Universal Robots PolyScope program: Example_palletsim_to_ur.urp

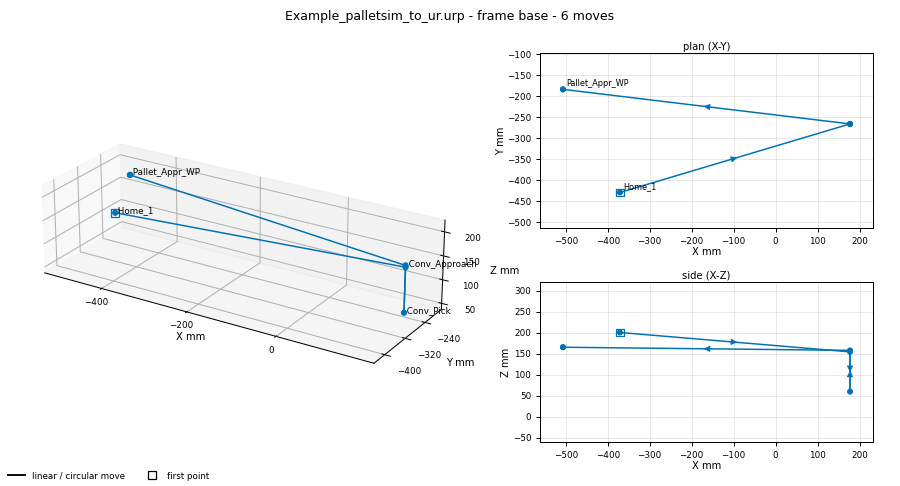
[picture p0: tool path of Example_palletsim_to_ur.urp in frame base, 6 of 9 moves have a stored position in this frame; points joined in program order, loops and branches not executed]
Program RidzwanPalletSoftware_3.2_Angle_URTrainingRoom (installation=default directory=/home/ur/ursim-current/programs createdIn=5.21.2 lastSavedIn=5.21.3 robotSerialNumber=20245799999)
Calibrated DH parameters: a=[0, -0.425, -0.3922, 0, 0, 0]; d=[0.1625, 0, 0, 0.1333, 0.0997, 0.0996]; alpha=[1.570796, 0, 0, 1.570796, -1.570796, 0]; deltaTheta=[0, 0, 0, 0, 0, 0]
InitVariablesNode
Robot Program (runOnlyOnce=false)
  Call Program_Execution
SubProgram -> Program_Execution
SubProgram Program_Execution (keepSynchronizedWithDisk=false)
  Folder Initial Instructions
    Popup Message (haltProgram=false message=Refer to the program Pop-up steps to complete the program, the following will be need/completed: <br><br> 1. IP_Address <br> 2. A.Palletizing and B. Conveyor <br> Approach and Exit waypoints <br> 3. Plane Feature  inputType=Text)
    Popup Warning (haltProgram=false message=*IMPORTANT* <br> <br> You will need to complete the instructions in all of the 'User Configuration' Folders found in the program inputType=Text)
    Popup Message (haltProgram=false message=First step will be to create a Plane Feature via the Installation tab. <br> <br> Make sure that the Origin is directly on the edge of the pallet. (Similar to visualization on Pallet Software program) inputType=Text)
  Folder Socket Configuration
    Folder User Configuration
      Popup Message (haltProgram=false message=Replace the X value below with the Manual IP_Address of the PC inputType=Text)
      PC_IPAddress := "192.168.56.5"
    Socket_Check := socket_open(PC_IPAddress,50000,socket_name="socket_0")
    asciiData := socket_read_ascii_float(8,"socket_0",timeout=0)
  MoveJ speed 60 deg/s, acceleration 80 deg/s^2 (useActiveTCP=true optimoveEnabled=false optiMoveSpeed=0.3 optiMoveAcceleration=0.09) feature=Base
    Waypoint Home_1: TCP in base x=-370.977 y=-429.532 z=201.159 mm, rx=-2.2649 ry=-2.1727 rz=-0.0079 rad; joints [-117.295, -100.067, -95.13, -75.173, 89.825, 65.225] deg; TCP offset x=0 y=0 z=176.9 mm, rx=0 ry=0 rz=0 rad
  'Conveyor'
  Folder Folder
    Folder Conveyor/Stationary Logic
      Set DigitalOutput pin=digital_out[2]; digitalValue=1
      Set AnalogOutput pin=analog_out[1]; analogValue=10
      Wait DigitalInput pin=digital_in[3]; digitalValue=1
      Wait Sleep waitTime=1
      Set DigitalOutput pin=digital_out[2]; digitalValue=0
      MoveL speed 250 mm/s, acceleration 1200 mm/s^2 (useActiveTCP=true optimoveEnabled=false optiMoveSpeed=0.3 optiMoveAcceleration=0.09) feature=Base
        Folder User Configuration
          Waypoint Conv_Approach: TCP in base x=177.389 y=-266.068 z=154.971 mm, rx=2.2689 ry=2.1729 rz=0 rad; joints [-31.936, -64.279, -132.627, -73.136, 89.936, 150.74] deg
          Waypoint Conv_Pick: TCP in base x=177.389 y=-266.068 z=60.124 mm, rx=2.2689 ry=2.1729 rz=0 rad; joints [-31.908, -72.825, -143.428, -53.79, 89.881, 150.729] deg
          Folder Gripper Logic
            URCap VG Grip (OnRobot, OnRobot A/S) dataModel(payload-weight=0.01, vg.grip.seek=false, Variable(key=on_return, variable(name=on_return)))
            Wait Sleep waitTime=0.25
          Waypoint Conv_Exit: TCP in base x=177.389 y=-266.068 z=158.52 mm, rx=2.2689 ry=2.1729 rz=0 rad; joints [-31.937, -64.094, -132.18, -73.767, 89.937, 150.74] deg
  'Pallet_Software'
  Folder Palletizing Software Logic
    boxCenterX := asciiData[3]
    boxCenterY := asciiData[4]
    AngleValue := asciiData[5]
    HeightValue := asciiData[6]
    MoveL speed 250 mm/s, acceleration 1200 mm/s^2 (useActiveTCP=true optimoveEnabled=false optiMoveSpeed=0.3 optiMoveAcceleration=0.09) feature=Base
      Folder User Configuration
        Waypoint Pallet_Appr_WP: TCP in base x=-506.661 y=-183.741 z=166.025 mm, rx=2.2689 ry=2.1729 rz=0 rad; joints [-145.856, -97.57, -103.549, -68.922, 89.882, 36.757] deg
      Wait Sleep waitTime=0.05
      tempVar := get_actual_tcp_pose()
      Pallet_App_Z := tempVar[2]
      Pallet_App_Rx := tempVar[3]
      Pallet_App_Ry := tempVar[4]
      Pallet_App_Rz := tempVar[5]
      CompilePoseRef := p[boxCenterX,boxCenterY,HeightValue,0,0,0]
      Folder User Configuration
        Execute_Pose := pose_trans(Plane_3,CompilePoseRef)
      tempVar := p[0,0,0,0,0,d2r(AngleValue)]
      Execute_Pose := p[Execute_Pose[0],Execute_Pose[1],Execute_Pose[2],Pallet_App_Rx,Pallet_App_Ry,Pallet_App_Rz]
      Execute_Pose := pose_trans(Execute_Pose,tempVar)
      Script: Pre_Execute_Pos=Execute_Pose
      Script: Pre_Execute_Pos[2]=Pallet_App_Z
      Waypoint Variable (Variable): variable=Pre_Execute_Pos
      Waypoint Variable (Variable): variable=Execute_Pose
      Folder User Configuration
        Folder Gripper Logic
          URCap VG Release (OnRobot, OnRobot A/S) dataModel(vg.channel.b=false)
          Wait Sleep waitTime=0.2
      Waypoint Variable (Variable): variable=Pre_Execute_Pos
      Folder User Configuration
        Waypoint Pallet_Exit_WP: TCP in base x=-506.661 y=-183.741 z=166.025 mm, rx=2.2689 ry=2.1729 rz=0 rad; joints [-145.856, -97.57, -103.549, -68.922, 89.882, 36.757] deg
  Wait Sleep waitTime=0.02
  Script: socket_send_string("NEXT", "socket_0")
